Staubli VAL3: COGNEX1.pjx

--- COGNEX1.pjx ---
Parameters version=s7.6 stackSize=5000 millimeterUnit=true
Program file=create.pgx
Program file=detection.pgx
Program file=getMaxNumOfPart.pgx
Program file=getObjectData.pgx
Program file=getObjectLatch.pgx
Program file=init.pgx
Program file=initvis.pgx
Program file=isDetected.pgx
Program file=kill.pgx
Program file=resetTask.pgx
Program file=sortObjects.pgx
Program file=start.pgx
Program file=stop.pgx
Data file=Cognex1.dtx
Library alias=ut path=Disk://Tracking/Tools/util/util.pjx autoload=true password=
Library alias=cam path=./cognexComm/cognexComm.pjx autoload=true password=
Library alias=sck path=Disk://Tracking/io/sockets/sockets.pjx autoload=true password=
Type name=object path=Disk://Tracking/Templates/object/object.pjx

--- initvis.pgx ---
program initvis(bool& x_bResult[] (dimensions=1))
  local bool l_bResult
begin
  // Initialize cognex communication library
  call cam:init()
  x_bResult=true
  clearBuffer(skVision)
  put("logging in to camera...")
  // log in to camera using socket cognex1 and return a handle in hCamTable
  //
  call cam:login(skVision,"admin","",hCamTable,l_bResult)
  if l_bResult
    putln("ok")
  else
    call cam:getErrorMessage(hCamTable,strError)
    putln("failed: "+strError)
    x_bResult=false
  endIf
  call cam:getOnline(hCamTable,l_bResult)
  if !l_bResult
    putln("Camera is not online")
    x_bResult=false
  endIf
end

--- sortObjects.pgx ---
program sortObjects(num x_nNumOfPart (dimensions=1))
  local num l_nI
  local num l_nMaxIndex
  local num l_nJ
  local num l_nMaxValue
begin
  // This program sorts the parts from the part with the largest X
  //  value to the smallest X value. This particular order is
  //  convenient when the orientation of the detection frame has the
  //  same orientation as the conveyor frame because the first part
  //  on the queue should be the first part to arrive into the
  //  tracking window.
  //
  //----------------------------------------------------------------
  //
  // Init variables
  l_nMaxIndex=0
  //
  // Sort parts from the largest X to the smallest X
  for l_nJ=0 to x_nNumOfPart-1
    // Find the largest X
    l_nMaxValue=-power(2,100)
    for l_nI=0 to x_nNumOfPart-1
      if trObjectPos[l_nI].x>l_nMaxValue and nObjectID[l_nI]>0
        l_nMaxValue=trObjectPos[l_nI].x
        l_nMaxIndex=l_nI
      endIf
    endFor
    // Copy largest
    oTempQueue[l_nJ].nID=nObjectID[l_nMaxIndex]
    oTempQueue[l_nJ].trTrsf=trObjectPos[l_nMaxIndex]
    oTempQueue[l_nJ].nLatchedValue=nLatchedValue[l_nMaxIndex]
    // Erase largest
    nObjectID[l_nMaxIndex]=-1
  endFor
  //
  // Copy sorted values
  for l_nI=0 to x_nNumOfPart-1
    nObjectID[l_nI]=oTempQueue[l_nI].nID
    trObjectPos[l_nI]=oTempQueue[l_nI].trTrsf
    nLatchedValue[l_nI]=oTempQueue[l_nI].nLatchedValue
  endFor
end
